FUNCTION_BLOCK SENSOR_SIMULATOR_V3
  {SET_ATTRIBUTE(OpcUa, DEVICE.SENSOR)}
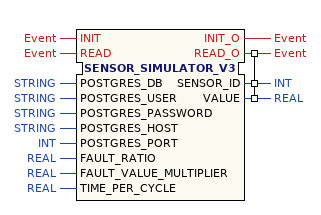
  EVENT_INPUT
    INIT;
    READ;
  END_EVENT
  EVENT_OUTPUT
    INIT_O;
    READ_O WITH VALUE, SENSOR_ID;
  END_EVENT
  VAR_INPUT
    POSTGRES_DB : STRING; {SET_ATTRIBUTE(OpcUa, Constant)}
    POSTGRES_USER : STRING; {SET_ATTRIBUTE(OpcUa, Constant)}
    POSTGRES_PASSWORD : STRING; {SET_ATTRIBUTE(OpcUa, Constant)}
    POSTGRES_HOST : STRING; {SET_ATTRIBUTE(OpcUa, Constant)}
    POSTGRES_PORT : INT; {SET_ATTRIBUTE(OpcUa, Constant)}
    FAULT_RATIO : REAL; {SET_ATTRIBUTE(OpcUa, Constant)}
    FAULT_VALUE_MULTIPLIER : REAL; {SET_ATTRIBUTE(OpcUa, Constant)}
    TIME_PER_CYCLE : REAL; {SET_ATTRIBUTE(OpcUa, Constant)}
  END_VAR
  VAR_OUTPUT
    SENSOR_ID : INT; {SET_ATTRIBUTE(OpcUa, Variable)}
    VALUE : REAL; {SET_ATTRIBUTE(OpcUa, Variable)}
  END_VAR
END_FUNCTION_BLOCK
